FUNCTION_BLOCK DEMO_Plant (* Filling-cell plant model for demos: needle travel, dosing, stoppering and inspection driven by the skills' Drive outputs; counts MoveDown/MoveUp shoot-through *)
  (* Standard: 61499-2 *)
  (* Version 2.0, 2026-09-27, Project contributors, Filling cell reference model *)
  PACKAGE fillingcell;
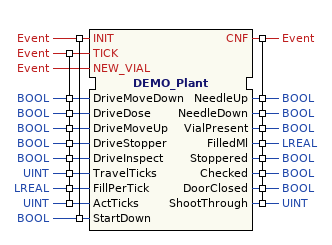
  EVENT_INPUT
    INIT WITH StartDown;
    TICK WITH DriveMoveDown, DriveDose, DriveMoveUp, DriveStopper, DriveInspect, TravelTicks, FillPerTick, ActTicks;
    NEW_VIAL;
  END_EVENT
  EVENT_OUTPUT
    CNF WITH NeedleUp, NeedleDown, VialPresent, FilledMl, Stoppered, Checked, DoorClosed, ShootThrough;
  END_EVENT
  VAR_INPUT
    DriveMoveDown : BOOL;
    DriveDose : BOOL;
    DriveMoveUp : BOOL;
    DriveStopper : BOOL;
    DriveInspect : BOOL;
    TravelTicks : UINT := 10;
    FillPerTick : LREAL := 0.02;
    ActTicks : UINT := 10;
    StartDown : BOOL;
  END_VAR
  VAR_OUTPUT
    NeedleUp : BOOL;
    NeedleDown : BOOL;
    VialPresent : BOOL;
    FilledMl : LREAL;
    Stoppered : BOOL;
    Checked : BOOL;
    DoorClosed : BOOL;
    ShootThrough : UINT;
  END_VAR
  VAR
    Position : UINT;
    StopTicks : UINT;
    InspTicks : UINT;
  END_VAR
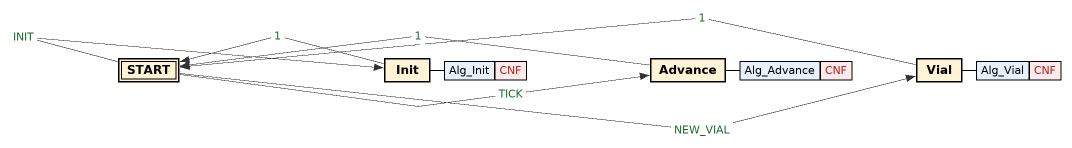
  EC_STATES
    START;
    Init : Alg_Init -> CNF;
    Advance : Alg_Advance -> CNF;
    Vial : Alg_Vial -> CNF;
  END_STATES
  EC_TRANSITIONS
    START TO Init := INIT;
    Init TO START := 1;
    START TO Advance := TICK;
    Advance TO START := 1;
    START TO Vial := NEW_VIAL;
    Vial TO START := 1;
  END_TRANSITIONS
  ALGORITHM Alg_Init IN ST:
Position := 0;
IF StartDown THEN Position := TravelTicks; END_IF;
VialPresent := TRUE;
DoorClosed := TRUE;
FilledMl := 0.0;
Stoppered := FALSE;
Checked := FALSE;
NeedleUp := Position = 0;
NeedleDown := Position >= TravelTicks;
  END_ALGORITHM
  ALGORITHM Alg_Advance IN ST:
IF DriveMoveDown AND DriveMoveUp THEN ShootThrough := ShootThrough + 1;
ELSIF DriveMoveDown AND (Position < TravelTicks) THEN Position := Position + 1;
ELSIF DriveMoveUp AND (Position > 0) THEN Position := Position - 1;
END_IF;
NeedleUp := Position = 0;
NeedleDown := Position >= TravelTicks;
IF DriveDose AND NeedleDown THEN FilledMl := FilledMl + FillPerTick; END_IF;
IF DriveStopper THEN StopTicks := StopTicks + 1; ELSE StopTicks := 0; END_IF;
IF StopTicks >= ActTicks THEN Stoppered := TRUE; END_IF;
IF DriveInspect THEN InspTicks := InspTicks + 1; ELSE InspTicks := 0; END_IF;
IF InspTicks >= ActTicks THEN Checked := TRUE; END_IF;
  END_ALGORITHM
  ALGORITHM Alg_Vial IN ST:
VialPresent := TRUE;
FilledMl := 0.0;
Stoppered := FALSE;
Checked := FALSE;
  END_ALGORITHM
END_FUNCTION_BLOCK
